(* IEC 61131-3 sources: ArfBotOS/Codesys-4/ArfBotOS.fbsdev/Application.iecapp^/FUN/group/FB_GroupHandler.fb.st^/P_GroupEnabled.prop.st^, 1 file *)

(* ---- Get.meth.st ---- *)
VAR
END_VAR

P_GroupEnabled := _GroupEnabled;
